Staubli VAL3: remGetPPS.pgx

program remGetPPS(string& sReturn[] (dimensions=1))
  local string sCmd
begin
  // Return the PPS status saved in the robot
  //
  logMsg("call remGetPPS")
  sCmd="GETPPS"
  call remGetnGlobal(nPPS,sCmd,sReturn)
end
